FUNCTION_BLOCK FB_UvLedModule EXTENDS FB_BasePrint IMPLEMENTS I_DeviceBase
VAR_INPUT
  IbReady                  AT%I* : BOOL;
END_VAR

VAR_OUTPUT
  ObEnableHigh             AT%Q* : BOOL;
  ObLowIntenseMode         AT%Q* : BOOL;
  ObDisableLeft            AT%Q* : BOOL;
  ObDisableRight           AT%Q* : BOOL;
  OnIntensitySetpoint      AT%Q* : WORD;  (*Setpoint for intensity control  [digit]*)
END_VAR

VAR
  _bActivate                     : BOOL;
  _sName                         : STRING := '';
  _StInkDefinition               : ST_INKDEFINITON;
END_VAR

VAR CONSTANT
  CnAnalogMinDigit               : DINT := 0;      (*Min value analog-output in digit*)
  CnAnalogMaxDigit               : DINT := 32767;  (*Max value analog-output in digit*)
  CnMinIntensitySetpoint         : DINT := 5;      (*Min setpoint for intensity control [%]*)
  CnMaxIntensitySetpoint         : DINT := 100;    (*Max setpoint for intensity control [%]*)
END_VAR

VAR PERSISTENT
  RbLowIntenseMode               : BOOL := FALSE;  (*Visu: set low intense mode*)
  RbDisableLeft                  : BOOL := FALSE;  (*Visu: disable left SLM*)
  RbDisableRight                 : BOOL := FALSE;  (*Visu: disable right SLM*)
  RnIntensitySetpoint            : DINT := 20;     (*Visu: setpoint for intensity control [%]*)
END_VAR

(*Set outputs*)
ObEnableHigh        := _bActivate;
ObLowIntenseMode    := RbLowIntenseMode;
ObDisableLeft       := RbDisableLeft;
ObDisableRight      := RbDisableRight;
OnIntensitySetpoint := DINT_TO_WORD(CnAnalogMaxDigit * RnIntensitySetpoint / 100);  (*Setpoint [digit]*)

METHOD mDisable : BOOL
_bActivate := FALSE;
END_METHOD

METHOD mEnable : BOOL
_bActivate := TRUE;
END_METHOD

{warning 'add property implementation'}
PROPERTY pActive : BOOL
GET
pActive := _bActivate;
END_GET
END_PROPERTY

{warning 'add property implementation'}
PROPERTY pErrorCode : INT
GET
END_GET
END_PROPERTY

PROPERTY pStInkDefinition : ST_INKDEFINITON
SET
_StInkDefinition := pStInkDefinition;
END_SET
END_PROPERTY

END_FUNCTION_BLOCK

(* stored: Version 1.1.0.1, ProductVersion 3.1.4024.3
   POU FB_UvLedModule: Id {bdfd1387-d538-43dc-9069-aa4a689b9f77}, SpecialFunc None
   Method mDisable: Id {585e4031-597f-4e92-b3a6-4290c11783d1}
   Method mEnable: Id {8e6de0ff-a87b-4556-8490-7c1428e8e1a4}
   Property pActive: Id {6b151028-6d9a-4a3c-b1da-f589e2879a49}
   Get Get: Id {62741bb7-e2f2-4b9c-8ba3-caf7aca10cbf}
   Property pErrorCode: Id {8d38e93d-26c6-4abc-908d-d3bbb0a546fc}
   Get Get: Id {e5910c2e-06db-429e-bd07-5fef50a89732}
   Property pStInkDefinition: Id {79cc3491-e246-4bad-a836-1d152c7a8e91}
   Set Set: Id {d422f218-8621-44b8-b46a-68b4b1d9c0ce} *)
